INTERFACE ITF_BaseLoggerElement_HMI_Connector_View

(*			
	RafalOS
	Rafał Osajda		09.06.2025		TC 4024.66
	Szuka czy ma zgłoszenie i zadanym ID jak tak to usuwa i zwraca true w przeciwnym razie zwraca false 
*)
METHOD PUBLIC EventAcknowledgeByID : BOOL
VAR_INPUT
	uiIDEvent				: UINT;
END_VAR
END_METHOD

(*			
	RafalOS
	Rafał Osajda		09.06.2025		TC 4024.66
	Szuka czy ma zgłoszenie i zadanym ID jak tak to usuwa i zwraca true w przeciwnym razie zwraca false 
*)
METHOD PUBLIC EventSetInactiveByID : BOOL
VAR_INPUT
	uiIDEvent				: UINT;
END_VAR
END_METHOD

METHOD PUBLIC GetCode : STRING
VAR_INPUT
END_VAR
END_METHOD

METHOD PUBLIC GetID : UINT
VAR_INPUT
END_VAR
END_METHOD

METHOD PUBLIC GetIdentyfier : ST_BaseElementIdentifier
VAR_INPUT
END_VAR
END_METHOD

METHOD PUBLIC GetName : ST_BaseLabel
VAR_INPUT
END_VAR
END_METHOD

METHOD PUBLIC GetType : E_BaseElementType
VAR_INPUT
END_VAR
END_METHOD

END_INTERFACE

(* stored: Version 1.1.0.1
   Itf ITF_BaseLoggerElement_HMI_Connector_View: Id {18066f33-5cce-0b8b-2b60-e60e4addcc02}
   Method EventAcknowledgeByID: Id {aa9672a4-c4e6-09f1-3f96-bba7e4c8f9c4}
   Method EventSetInactiveByID: Id {dcdbc491-0072-0718-3d2c-19591fbbe90d}
   Method GetCode: Id {f5cf3e5c-088f-0e43-06f5-119997559e59}
   Method GetID: Id {6d80811c-c1cb-062f-0769-541a69ee6d76}
   Method GetIdentyfier: Id {ac6e2f1d-ef73-047b-0178-a3d1abb02eb3}
   Method GetName: Id {8b277639-3747-0d1b-09fd-1b4180f8280b}
   Method GetType: Id {39784064-3fc4-0e64-092d-21b915a721a1} *)
